{attribute 'qualified_only'}
VAR_GLOBAL
    
    SAFETYRUN AT %Q* : BOOL := TRUE;
    ERRACK AT %Q* : BOOL;
    MUTE_LC AT %Q* : BOOL := FALSE;
    MUTE_ENABLING AT %Q* : BOOL := FALSE;
    UNMUTE_ENABLING AT %Q* : BOOL;
    NORMALMODE_FB_STATE AT %I*: USINT;
END_VAR

(* stored: Version 1.1.0.1, ProductVersion 3.1.4024.5
   GVL GVL_Safety: Id {f8271d8d-c0b2-4e7b-82c7-58623e649ac4} *)
